FUNCTION IsValidInterface : BOOL
VAR_INPUT
	ip : I_Base;
END_VAR

IsValidInterface := (ip <> 0);

END_FUNCTION

(* stored: Version 1.1.0.1, ProductVersion 3.1.4026.18
   POU IsValidInterface: Id {f18c148e-a18a-4c4d-b322-3d8ac753f575}, SpecialFunc None *)
